{attribute 'linkalways'} 
{attribute 'no_explicit_call' := 'This FB is a CLASS and must be accessed using methods or properties'}
{attribute 'enable_dynamic_creation'}
FUNCTION_BLOCK _TcVnVector4_SINT EXTENDS AliasDatatypeBase
VAR
	localData : TcVnVector4_SINT;
	activeData : REFERENCE TO TcVnVector4_SINT REF= localData;
	aliasBaseDatatype : _Array0to3OfSINT;
END_VAR

PROPERTY PUBLIC Address : PVOID
GET
Address := ADR(activeData);
END_GET
END_PROPERTY

METHOD PUBLIC ClearReference
VAR_INPUT
END_VAR
activeData REF= localData;
SetBaseDatatypeReference();
END_METHOD

METHOD PUBLIC Clone : I_Datatype
VAR
    pClone : POINTER TO _TcVnVector4_SINT;
END_VAR
pClone := __NEW(_TcVnVector4_SINT);
Clone := pClone^;
END_METHOD

METHOD FB_init : BOOL
VAR_INPUT
	bInitRetains : BOOL; // if TRUE, the retain variables are initialized (warm start / cold start)
	bInCopyCode : BOOL;  // if TRUE, the instance afterwards gets moved into the copy code (online change)
	//InitialValue : <type>; // if possible, not all values can be initialized
END_VAR
//localData := InitialValue; // if possible, not all values can be initialized
SetBaseDatatypeReference();
AddBaseDatatype(aliasBaseDatatype);
END_METHOD

PROPERTY PUBLIC Identifier : T_MAXSTRING
GET
Identifier := 'TcVnVector4_SINT';
END_GET
END_PROPERTY

METHOD PUBLIC MakeReferenceTo
VAR_INPUT
	ReferenceTarget : REFERENCE TO TcVnVector4_SINT;
END_VAR
activeData REF= ReferenceTarget;
SetBaseDatatypeReference();
END_METHOD

METHOD PROTECTED SetBaseDatatypeReference
VAR_INPUT
END_VAR
aliasBaseDatatype.MakeReferenceTo(activeData);
END_METHOD

PROPERTY PUBLIC Size : UDINT
GET
Size := SIZEOF(activeData);
END_GET
END_PROPERTY

METHOD TryMakeReferenceTo : BOOL
VAR_INPUT
	Target : I_Datatype;
END_VAR
VAR
	pTargetData : POINTER TO TcVnVector4_SINT;
END_VAR
IF NOT IsEquivalentTo(Target) THEN
	RETURN;
END_IF

pTargetData := Target.Address;
activeData REF= pTargetData^;
SetBaseDatatypeReference();
TryMakeReferenceTo := TRUE;
END_METHOD

PROPERTY PUBLIC Value : REFERENCE TO TcVnVector4_SINT
GET
Value REF= activeData;
END_GET
END_PROPERTY

END_FUNCTION_BLOCK

(* stored: Version 1.1.0.1, ProductVersion 3.1.4024.13
   POU _TcVnVector4_SINT: Id {fc7c716b-168c-0a1d-004c-ed3e566a9f04}, SpecialFunc None
   Folder Core: Id {3c445252-ac2b-0c0a-16de-82443933c0af}
   Folder Protected: Id {e876d0fa-6a81-0c69-3a8d-d1aa3e5e9945}
   Folder Customize: Id {322e185d-f099-0110-0b23-a62e7d0d7b83}
   Folder Constructor: Id {cbcbf26f-fa0d-0395-0af3-987c0577b6cb}
   Property Address: Id {43a0d8c8-be2d-036b-1008-577393d4a087}
   Get Get: Id {2c475e9e-a75c-0b2f-0958-752136311717}
   Method ClearReference: Id {1715f43a-ea2f-0074-1c6c-0402ef106ce0}
   Method Clone: Id {e2ea59bc-ed48-0373-1635-e61392537a2b}
   Method FB_init: Id {585f44a6-188d-0945-04e4-a7ac7e778f4c}
   Property Identifier: Id {f2717a3d-1acf-0301-0dc7-aa8cc63f6804}
   Get Get: Id {0c4fed7d-a06b-0d8b-00b7-838fbb964516}
   Method MakeReferenceTo: Id {24600136-88ae-0f3e-3302-caa091c33ce4}
   Method SetBaseDatatypeReference: Id {6d2562f8-55fd-08f5-31b5-40a45da5f10f}
   Property Size: Id {d3895ab0-1bd7-0a86-00aa-c851d55258d4}
   Get Get: Id {5048c905-4023-0b00-0455-30597de3aa26}
   Method TryMakeReferenceTo: Id {733de445-d532-0c72-0615-384614bf17ab}
   Property Value: Id {6b5ff6be-843d-07b9-1b8c-a1104e0d5d97}
   Get Get: Id {ede34ace-75e6-0888-0219-872dd7ec58b7} *)
